// Mitsubishi GX Works2 project: 开关简单自锁   PLC: FX3U/FX3UC

PROGRAM MAIN
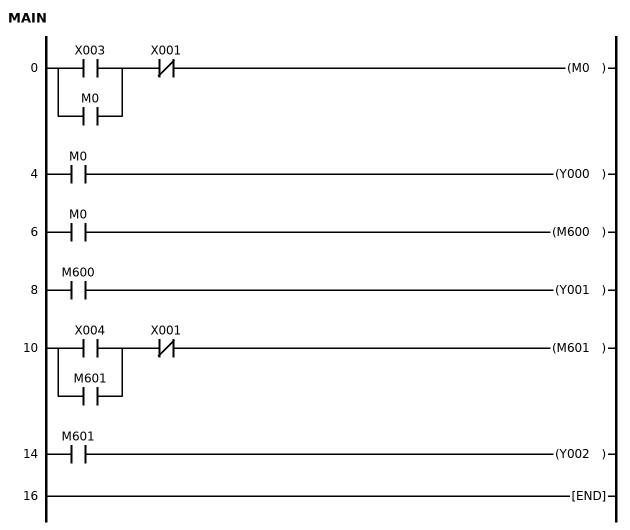
0     LD      X003
      OR      M0
      ANI     X001
      OUT     M0
4     LD      M0
      OUT     Y000
6     LD      M0
      OUT     M600
8     LD      M600
      OUT     Y001
10    LD      X004
      OR      M601
      ANI     X001
      OUT     M601
14    LD      M601
      OUT     Y002
16    END
END_PROGRAM
